// TIA Portal V20 export
FUNCTION_BLOCK "RealFbName"   // FB2, LAD
   VAR_INPUT
      Enable : Bool;
   END_VAR
BEGIN
END_FUNCTION_BLOCK
